// TIA Portal V19 export
DATA_BLOCK "Panel"   // DB1070
{ S7_Optimized_Access := 'TRUE' }
// stored: AutoNumber false, MemoryReserve 100
   VAR RETAIN
      IW : Struct   // Analogwerte
         "LF_CM01.BN01" : Real;   // Leitfähigkeit Bypass Filterpumpe
         "LF_CM01.BN02" : Real;   // Leitfähigkeit Düsen Umwälzung
         "LF_CM02.BN03" : Real;   // Leitfähigkeit Bypass Filterpumpe
         "LF_CM02.BN04" : Real;   // Leitfähigkeit Düsen Umwälzung
         "p_HQ01.BP01" : Real;   // Druck Beutelfiltergehäuse
         "p_HQ02.BP02" : Real;   // Druck Beutelfiltergehäuse
         "p_CM01.BP03" : Real;   // Druck Filterpumpe
         "p_CM01.BP04" : Real;   // Druck Umwälzpumpe
         "p_CM03.BP05" : Real;   // Druck Umwäzpumpe
         "p_CM02.BP06" : Real;   // Druck Filterpumpe
         "p_CM02.BP07" : Real;   // Druck Umwälzpumpe
         "p_CM04.BP08" : Real;   // Druck Umwäzpumpe
         "p_CM05.BP09" : Real;   // Druck Pumpe Entleerung Sammeltank
         "Dfl_GP01.BF01" : Real;   // Durchfluss Versorgung Frischsäure
         "Dfl_GP02.BF02" : Real;   // Durchfluss Entsorgung Altsäure
         "Niv_GP01.BL30" : Real;   // Füllstand Versorgung Frischsäure
         "Niv_GP02.BL31" : Real;   // Füllstand Entsorgung Altsäure
         pH_BE : Real;   // SRM_Auf_BG-QM43
      END_STRUCT;
      Deckel : Struct   // Deckel Säurebecken
         CM01 : Struct
            Auto : Bool;
            Hand : Bool;
            Tipp : Bool;
            links_auf : Bool;
            links_zu : Bool;
            rechts_auf : Bool;
            rechts_zu : Bool;
            SRM_links_auf : Bool;
            SRM_links_zu : Bool;
            SRM_rechts_auf : Bool;
            SRM_rechts_zu : Bool;
            S_links_auf : Bool;   // CM01.BG01
            S_links_zu : Bool;   // CM01.BG02
            S_rechts_auf : Bool;   // CM01.BG03
            S_rechts_zu : Bool;   // CM01.BG04
            Ist_Pos_links : Int;   // 0% = auf; 100% = zu
            Ist_Pos_rechts : Int;   // 0% = auf; 100% = zu
         END_STRUCT;
         CM02 : Struct
            Auto : Bool;
            Hand : Bool;
            Tipp : Bool;
            links_auf : Bool;
            links_zu : Bool;
            rechts_auf : Bool;
            rechts_zu : Bool;
            SRM_links_auf : Bool;
            SRM_links_zu : Bool;
            SRM_rechts_auf : Bool;
            SRM_rechts_zu : Bool;
            S_links_auf : Bool;   // CM02.BG01
            S_links_zu : Bool;   // CM02.BG02
            S_rechts_auf : Bool;   // CM02.BG03
            S_rechts_zu : Bool;   // CM02.BG04
            Ist_Pos_links : Int;   // 0% = auf; 100% = zu
            Ist_Pos_rechts : Int;   // 0% = auf; 100% = zu
         END_STRUCT;
      END_STRUCT;
      RT : Struct   // Schnelllauftor
         K_Auto : Bool;   // Knauf Auto
         T_auf : Bool;   // Taste RT auf
         T_zu : Bool;   // Taste RT zu
         MSS_ok : Bool;   // Motorschutzschalter o.k.
         S_offen : Bool;   // Schnelllauftor offen
         S_geschlossen : Bool;   // Schnelllauftor geschlossen
         ok : Bool;   // Schnelllauftor o.k.
         Status : USInt;
      END_STRUCT;
      Ventilator : Struct   // FU[7]
         Ein : Bool;
         Auto : Bool;
         laeuft : Bool;
         betriebsbereit : Bool;
         Stoerung : Bool;
         Status : USInt;
         SW_Hand : Int;   // [%]
         SW_Auto_AZ : Int;   // [%]
         SW_Auto_aAZ : Int;   // [%]
         speed : Int;   // [%]
      END_STRUCT;
      CM01 : Struct   // HF-Becken 1
         Betrieb : Bool;
         Wartung : Bool;
         Niv_TGS : Bool;   // BL04
         Niv_Min : Bool;   // BL03
         Niv_max : Bool;   // BL02
         Niv_Uel : Bool;   // BL01
         NSP_Auto : Bool;
         GW_LF_FP : Bool;   // BN01
         GW_LF_UP : Bool;   // BN02
         GW_p_FP : Bool;   // BP03
         GW_p_UP : Bool;   // BP04
         Niv_Proz : USInt;
         Sollwert_LF : Real;   // Dosierung
         Dosierung_LF : Bool;   // 0 = WT, 1= LF
      END_STRUCT;
      CM02 : Struct   // HF-Becken 2
         Betrieb : Bool;
         Wartung : Bool;
         Niv_TGS : Bool;   // BL11
         Niv_Min : Bool;   // BL10
         Niv_max : Bool;   // BL09
         Niv_Uel : Bool;   // BL08
         NSP_Auto : Bool;
         GW_LF_FP : Bool;   // BN03
         GW_LF_UP : Bool;   // BN04
         GW_p_FP : Bool;   // BP06
         GW_p_UP : Bool;   // BP07
         Niv_Proz : USInt;
         Sollwert_LF : Real;   // Dosierung
         Dosierung_LF : Bool;   // 0 = WT, 1= LF
      END_STRUCT;
      CM03 : Struct   // Spülbecken 1
         Betrieb : Bool;
         Wartung : Bool;
         Niv_TGS : Bool;   // BL07
         Niv_Min : Bool;   // BL06
         GW_p_UP : Bool;   // BP05
         Niv_Proz : USInt;
         SPR_Auto : Bool;
         SPR_Start_Test : Bool;
         SPR_Stopp_Test : Bool;
         SPR_Zeit_Test : Int;
      END_STRUCT;
      CM04 : Struct   // Spülbecken 2
         Betrieb : Bool;
         Wartung : Bool;
         Niv_TGS : Bool;   // BL14
         Niv_Min : Bool;   // BL13
         GW_p_UP : Bool;   // BP08
         Niv_Proz : USInt;
         SPR_Auto : Bool;
         SPR_Start_Test : Bool;
         SPR_Stopp_Test : Bool;
         SPR_Zeit_Test : Int;
         NSP_Auto : Bool;
         NSP_Zeit : Int;   // pro Korb
         NSP_Start_Test : Bool;
         NSP_Stopp_Test : Bool;
         NSP_Zeit_Tes : Int;
      END_STRUCT;
      CM05 : Struct   // Abwassersammler
         Betrieb : Bool;
         Wartung : Bool;
         Niv_TGS : Bool;   // BL03
         Niv_Min : Bool;   // BL02
         Niv_max : Bool;   // BL01
         Niv_Uel : Bool;   // BL05
         AWA_Bereit : Bool;
         Frg_Abpumpen : Bool;
         GW_p_Pu : Bool;   // BP09
         Niv_Proz : USInt;
      END_STRUCT;
      HQ01 : Struct   // Filtereinheit
         Niv_Leckage : Bool;   // BL05
         GW_p_FG : Bool;   // BP01
         S_FG_zu : Bool;   // BG06
         S_Dkl_FG_li : Bool;   // BG07
         S_Dkl_FG_re : Bool;   // BG08
         Quitt_FW : Bool;
         Quitt_FW_erlaubt : Bool;
         WarnGr_FW : Real;
         Wechsel_FW : Real;
      END_STRUCT;
      HQ02 : Struct   // Filtereinheit
         Niv_Leckage : Bool;   // BL12
         GW_p_FG : Bool;   // BP02
         S_FG_zu : Bool;   // BG09
         S_Dkl_FG_li : Bool;   // BG10
         S_Dkl_FG_re : Bool;   // BG1
         Quitt_FW : Bool;
         Quitt_FW_erlaubt : Bool;
         WarnGr_FW : Real;
         Wechsel_FW : Real;
      END_STRUCT;
      GP01 : Struct   // HF-Versorgung
         Versorgung : Bool;
         Entsorgung : Bool;
         Niv_leer : Bool;   // BL17
         Niv_max : Bool;   // BL20
         IBC_vorhanden : Bool;   // BG21
         Tür_zu_vorn : Bool;   // BG44
         Tür_zu_seitlich : Bool;   // BG43
         LS_PuSu : Bool;   // BL18
         LS_Pumpe : Bool;   // BL15
         LS_Doppelrohr_BL19 : Bool;   // BL19
         LS_PFA_Übergang : Bool;   // BL16
         LS_Uml_Tunnel : Bool;   // BL34
         Niv_Proz : USInt;
         Status : USInt;
      END_STRUCT;
      GP02 : Struct   // HF-Entsorgung
         Versorgung : Bool;
         Entsorgung : Bool;
         Niv_leer : Bool;   // BL24
         Niv_max : Bool;   // BL23
         IBC_vorhanden : Bool;   // BG22
         Tür_zu_seitlich : Bool;   // BG45
         LS_PuSu : Bool;   // BL18
         LS_Pumpe : Bool;   // BL27
         LS_PFA_Übergang : Bool;   // BL25
         LS_Doppelrohr_BL26 : Bool;   // BL26
         LS_Doppelschlauch_BL32 : Bool;   // BL32
         LS_Doppelschlauch_BL33 : Bool;   // BL33
         Niv_Proz : USInt;
         Status : USInt;
      END_STRUCT;
      Havarie_GP0x : Struct
         Soll_Spuelen_CM0x : Real;   // [l]
         Ist_Spuelen_CM0x : Real;   // [l]
      END_STRUCT;
      CL0x : Struct
         "LS_CL01.BL28" : Bool;   // Leckage OK Übergabestation CL01 CL01.BL28
         "LS_CL02.BL29" : Bool;   // Leckage OK Pumpensumpf Säurebecken CL02 CL02.BL29
         Niv_Proz_CL01 : USInt;
         Niv_Proz_CL02 : USInt;
      END_STRUCT;
      FP_CM01 : Struct   // GP01
         Ein : Bool;
         Auto : Bool;
         Bedienung_Erlaubt : Bool;
         betriebsbereit : Bool;
         Stoerung : Bool;
         Sp_Ventil : Struct
            Sollzeit : Int;   // [s]
            Restzeit : Int;   // [s]
         END_STRUCT;
         Sp_Filter : Struct
            Zeit_leeren_Saure : Int;   // [s]
            Zeit_leeren_CM05 : Int;
            Zeit_Spülen : Int;   // [s]
            Wartezeit : Int;   // [s]
            Zeit_füllen : Int;   // [s]
            Restzeit : Int;   // [s]
         END_STRUCT;
         Drucktest_Pumpe : Struct
            Solldruck : Real;
            Sollzeit : Int;
            Restzeit : Int;
            Schritt : USInt;
         END_STRUCT;
         Drucktest_Filter : Struct
            Solldruck : Real;
            Sollzeit : Int;
            Restzeit : Int;
            Schritt : USInt;
         END_STRUCT;
         BA : USInt;   // 0=normal, 1=Filterwechsel, 2=Spülen
         Status : USInt;
         Status_FW : USInt;
         SW_Hand : Int;   // [%]
         SW_Auto_AZ : Int;   // [%]
         SW_Auto_aAZ : Int;   // [%]
         speed : Int;   // [%]
      END_STRUCT;
      UP_CM01 : Struct   // GP02
         Ein : Bool;
         Auto : Bool;
         Bedienung_Erlaubt : Bool;
         betriebsbereit : Bool;
         Stoerung : Bool;
         Sp_Ventil : Struct
            Sollzeit : Int;   // [s]
            Restzeit : Int;   // [s]
         END_STRUCT;
         Drucktest : Struct
            Solldruck : Real;
            Sollzeit : Int;
            Restzeit : Int;
            Schritt : USInt;
         END_STRUCT;
         BA : USInt;   // 0=normal, 1=Ents GP02, 2= Ents GP01, 3=Ents. CM05, 4=Spülen
         Status : USInt;
         SW_Hand : Int;   // [%]
         SW_Auto_AZ : Int;   // [%]
         SW_Auto_aAZ : Int;   // [%]
         speed : Int;   // [%]
      END_STRUCT;
      UP_CM03 : Struct   // GP03
         Ein : Bool;
         Auto : Bool;
         betriebsbereit : Bool;
         Bedienung_Erlaubt : Bool;
         Stoerung : Bool;
         Sp_Ventil : Struct
            Sollzeit : Int;   // [s]
            Restzeit : Int;   // [s]
         END_STRUCT;
         Drucktest : Struct
            Solldruck : Real;
            Sollzeit : Int;
            Restzeit : Int;
            Schritt : USInt;
         END_STRUCT;
         BA : USInt;   // 0=normal, 1=Ents. CM05, 2=Spülen
         Status : USInt;
         SW_Hand : Int;   // [%]
         SW_Auto_AZ : Int;   // [%]
         SW_Auto_aAZ : Int;   // [%]
         speed : Int;   // [%]
      END_STRUCT;
      FP_CM02 : Struct   // GP04
         Ein : Bool;
         Auto : Bool;
         Bedienung_Erlaubt : Bool;
         betriebsbereit : Bool;
         Stoerung : Bool;
         Sp_Ventil : Struct
            Sollzeit : Int;   // [s]
            Restzeit : Int;   // [s]
         END_STRUCT;
         Sp_Filter : Struct
            Zeit_leeren_Saure : Int;   // [s]
            Zeit_leeren_CM05 : Int;
            Zeit_Spülen : Int;   // [s]
            Wartezeit : Int;   // [s]
            Zeit_füllen : Int;   // [s]
            Restzeit : Int;   // [s]
         END_STRUCT;
         Drucktest_Pumpe : Struct
            Solldruck : Real;
            Sollzeit : Int;
            Restzeit : Int;
            Schritt : USInt;
         END_STRUCT;
         Drucktest_Filter : Struct
            Solldruck : Real;
            Sollzeit : Int;
            Restzeit : Int;
            Schritt : USInt;
         END_STRUCT;
         BA : USInt;   // 0=normal, 1=Filterwechse, 2=Spülen
         Status : USInt;
         Status_FW : USInt;
         SW_Hand : Int;   // [%]
         SW_Auto_AZ : Int;   // [%]
         SW_Auto_aAZ : Int;   // [%]
         speed : Int;   // [%]
      END_STRUCT;
      UP_CM02 : Struct   // GP05
         Ein : Bool;
         Auto : Bool;
         Bedienung_Erlaubt : Bool;
         betriebsbereit : Bool;
         Stoerung : Bool;
         Sp_Ventil : Struct
            Sollzeit : Int;   // [s]
            Restzeit : Int;   // [s]
         END_STRUCT;
         Drucktest : Struct
            Solldruck : Real;
            Sollzeit : Int;
            Restzeit : Int;
            Schritt : USInt;
         END_STRUCT;
         BA : USInt;   // 0=normal, 1=Ents GP02, 2= Ents GP01, 3=Ents. CM05, 4=Spülen
         Status : USInt;
         SW_Hand : Int;   // [%]
         SW_Auto_AZ : Int;   // [%]
         SW_Auto_aAZ : Int;   // [%]
         speed : Int;   // [%]
      END_STRUCT;
      UP_CM04 : Struct   // GP06
         Ein : Bool;
         Auto : Bool;
         betriebsbereit : Bool;
         Bedienung_Erlaubt : Bool;
         Stoerung : Bool;
         Sp_Ventil : Struct
            Sollzeit : Int;   // [s]
            Restzeit : Int;   // [s]
         END_STRUCT;
         Drucktest : Struct
            Solldruck : Real;
            Sollzeit : Int;
            Restzeit : Int;
            Schritt : USInt;
         END_STRUCT;
         BA : USInt;   // 0=normal, 1=Ents. CM05, 2=Spülen
         Status : USInt;
         SW_Hand : Int;   // [%]
         SW_Auto_AZ : Int;   // [%]
         SW_Auto_aAZ : Int;   // [%]
         speed : Int;   // [%]
      END_STRUCT;
      Pu_CM05 : Struct   // GP11
         Ein : Bool;
         Auto : Bool;
         Bedienung_Erlaubt : Bool;
         Sp_Ventil : Struct
            Sollzeit : Int;   // [s]
            Restzeit : Int;   // [s]
         END_STRUCT;
         Drucktest : Struct
            Solldruck : Real;
            Sollzeit : Int;
            Restzeit : Int;
            Schritt : USInt;
         END_STRUCT;
         BA : USInt;   // 0=Entl., 1=Kreislauf, 2=Spülen
         Status : USInt;
      END_STRUCT;
      Pu_CL01 : Struct   // GP08
         Ein : Bool;
         Auto : Bool;
         Bedienung_Erlaubt : Bool;
         Sp_Ventil : Struct
            Sollzeit : Int;   // [s]
            Restzeit : Int;   // [s]
         END_STRUCT;
         BA : USInt;   // 0=Ents. CM05, 1=Spülen
         Status : USInt;
      END_STRUCT;
      Pu_CL02 : Struct   // GP09
         Ein : Bool;
         Auto : Bool;
         Bedienung_Erlaubt : Bool;
         Sp_Ventil : Struct
            Sollzeit : Int;   // [s]
            Restzeit : Int;   // [s]
         END_STRUCT;
         BA : USInt;   // 0=Ents. CM05, 1=Spülen
         Status : USInt;
      END_STRUCT;
      Pu_Entl_GP01 : Struct   // GP12
         Ein : Bool;
         Auto : Bool;
         Bedienung_Erlaubt : Bool;
         Sp_Ventil : Struct
            Sollzeit : Int;   // [s]
            Restzeit : Int;   // [s]
         END_STRUCT;
         BA : USInt;   // 0=Ents. CM05, 1=Spülen
         Status : USInt;
      END_STRUCT;
      Pu_Vers_GP01 : Struct   // GP13
         Ein : Bool;
         Auto : Bool;
         Bedienung_Erlaubt : Bool;
         Sp_Ventil : Struct
            Sollzeit : Int;   // [s]
            Restzeit : Int;   // [s]
         END_STRUCT;
         BA : USInt;   // 0=Vers UVGP01, 1=Ents CM05, 2=Spülen
         Status : USInt;
      END_STRUCT;
      Pu_Entl_GP02 : Struct   // GP07
         Ein : Bool;
         Auto : Bool;
         Bedienung_Erlaubt : Bool;
         Sp_Ventil : Struct
            Sollzeit : Int;   // [s]
            Restzeit : Int;   // [s]
         END_STRUCT;
         BA : USInt;   // 0=Ents. CM05, 1=Spülen
         Status : USInt;
      END_STRUCT;
      Pu_Vers_GP02 : Struct   // GP10
         Ein : Bool;
         Auto : Bool;
         Bedienung_Erlaubt : Bool;
         Sp_Ventil : Struct
            Sollzeit : Int;   // [s]
            Restzeit : Int;   // [s]
         END_STRUCT;
         BA : USInt;   // 0=Vers UVGP01, 1=Ents CM05,2= Spülen
         Status : USInt;
      END_STRUCT;
      Pu_Entleeren : Struct   // GP14
         Ein : Bool;
         Status : USInt;
      END_STRUCT;
      Ventil : Struct   // 0 = Aus, 1= aktiv, 2=Störung
         "CM01.QM18" : USInt;   // Eingang Saugleitung Filterpumpe GP01 Säure 01 CM01.QM18
         "CM01.QM19" : USInt;   // Eingang Spülleitung Filterpumpe GP01 Säure 01 CM01.QM19
         "CM01.QM20" : USInt;   // Eingang Spülleitung Umwälzpumpe GP02 Säure 01 CM01.QM20
         "HQ01.QM21" : USInt;   // EingangSäureleitung Filtereinheit HQ02 Säure 01 CM01.QM21
         "HQ01.LV01" : USInt;   // Entlüftungs-/ Überdruckventil Beutelfilter Säure 01 HQ01.LV01
         "HQ01.QM22" : USInt;   // Eingang Spülleitung Filtereinheit HQ01 Säure 01 HQ01.QM22
         "HQ01.QM23" : USInt;   // Ausgang Säureleitung Filtereinheit HQ01 Säure 01 HQ01.QM23
         "HQ01.QM24" : USInt;   // Ausgang Spülleitung Filtereinheit HQ01 Säure 01 zu Sammeltank HQ01.QM24
         "CM01.QM25" : USInt;   // Eingang Saugleitung Umwälzpumpe GP02 Säure 01 CM01.QM25
         "CM01.QM26" : USInt;   // Ausgang Druckleitung Umwälzpumpe GP02 Säure 01 CM01.QM26
         "CM01.QM27" : USInt;   // Ausgang Spülleitung Umwälzpumpe GP02 Säure 01 zu Sammeltank CM01.QM27
         "CM03.QM33" : USInt;   // Eingang Saugleitung Umwälzpumpe GP03 Spülbecken 1 CM03.QM33
         "CM03.QM34" : USInt;   // Ausgang Druckleitung Umwälzpumpe GP03 Spülbecken 1 CM03.QM34
         "CM03.QM36" : USInt;   // Eingang Spülleitung Umwälzpumpe GP03 Spülbecken 1 CM03.QM36
         "CM03.QM37" : USInt;   // Ausgang Spülleitung Umwälzpumpe GP03 Spülbecken 1 CM03.QM37
         "CM02.QM55" : USInt;   // Eingang Saugleitung Filterpumpe GP04 Säure 02 CM02.QM55
         "CM02.QM56" : USInt;   // Eingang Spülleitung Filterpumpe GP04 Säure 02 CM02.QM56
         "CM02.QM57" : USInt;   // Eingang Spülleitung Umwälzpumpe GP05 Säure 02 CM02.QM57
         "HQ02.QM58" : USInt;   // Eingang Spülleitung Filtereinheit HQ02 Säure 02 CM02.QM58
         "HQ02.LV02" : USInt;   // Entlüftungs-/ Überdruckventil Beutelfilter Säure 02 HQ02.LV02
         "HQ02.QM59" : USInt;   // Eingang Säureleitung Filtereinheit HQ02 Säure 02 HQ02.QM59
         "HQ02.QM60" : USInt;   // Ausgang Säureleitung Filtereinheit HQ02 Säure 02 HQ02.QM60
         "HQ02.QM61" : USInt;   // Ausgang Spülleitung Filtereinheit HQ02 Säure 02 zu Sammeltank HQ02.QM61
         "CM02.QM62" : USInt;   // Eingang Saugleitung Umwälzpumpe GP05 Säure 02 CM02.QM62
         "CM02.QM63" : USInt;   // Ausgang Druckleitung Umwälzpumpe GP05 Säure 02 CM02.QM63
         "CM02.QM64" : USInt;   // Ausgang Spülleitung Umwälzpumpe GP05 Säure 02 zu Sammeltank CM02.QM64
         "CM04.QM72" : USInt;   // Eingang Saugleitung Umwälzpumpe GP06 Spülbecken 2 CM04.QM72
         "CM04.QM73" : USInt;   // Ausgang Druckleitung Umwälzpumpe GP06 Spülbecken 2 CM04.QM73
         "CM04.QM75" : USInt;   // Eingang Spülleitung Umwälzpumpe GP06 Spülbecken 2 CM04.QM75
         "CM04.QM76" : USInt;   // Ausgang Spülleitung Umwälzpumpe GP06 Spülbecken 2 CM04.QM76
         "CM04.QM77" : USInt;   // Frischwasserzufuhr Nachdosierung Spülbecken 2 CM04.QM77
         "CL01.QM51" : USInt;   // Zuleitung VE-Wasser-Spülung Pumpe GP08 CL01.QM51
         "CL02.QM52" : USInt;   // Zuleitung VE-Wasser-Spülung Pumpe GP09 CL02.QM52
         "CM05.QM61" : USInt;   // Saugseite Förderpumpe Entleerung GP11 Sammeltank CM05 CM05.QM61
         "CM05.QM62" : USInt;   // Eingang Spülleitung Förderpumpe GP11 Sammeltank CM05 CM05.QM62
         "CM05.QM63" : USInt;   // Ausgang Spülleitung Förderpumpe GP11 Sammeltank CM05 CM05.QM63
         "CM05.QM64" : USInt;   // Druckseite Förderpumpe Entleerung GP11 Sammeltank CM05 CM05.QM64
         "CM03.QM35" : USInt;   // VE-Wasserleitung Spritzregister Spülbecken 1 CM03.QM35
         "CM04.QM74" : USInt;   // VE-Wasserleitung Spritzregister Spülbecken 2 CM04.QM74
         "GP01.QM14" : USInt;   // PFA Schlauchleitung Anbindung IBC Quick Connect Entsorgung GP01.QM14
         "GP01.QM15" : USInt;   // Eingang Saugleitung Membranpumpe GP13 Versorgung Frischsäure GP01.QM15
         "GP01.QM16" : USInt;   // Eingang Spülleitung Membranpumpe GP13 Versorgung Frischsäure GP01.QM16
         "GP01.QM17" : USInt;   // Ausgang Spülleitung Membranpumpe GP13 Versorgung zu Sammeltank GP01.QM17
         "GP01.QM18" : USInt;   // Ausgang Druckleitung Membranpumpe GP13 Versorgung zu UV-GP01 GP01.QM18
         "GP01.QM19" : USInt;   // Verriegelung UV-GP01 Versorgungsleitung zu Säure CM2 GP01.QM19
         "GP01.QM20" : USInt;   // Verriegelung UV-GP01 Versorgungsleitung zu Säure CM1 GP01.QM20
         "GP01.QM21" : USInt;   // Verriegelung UV-GP01 Versorgungsleitung zur Entsorgung GP02 GP01.QM21
         "GP01.QM22" : USInt;   // Verriegelung UV-GP01 Versorgungsleitung zur Versorgung GP01 GP01.QM22
         "GP01.QM23" : USInt;   // VE-Wasser-Spülung GP12 zu Auffangwanne GP01.QM23
         "GP02.QM37" : USInt;   // VE-Wasser-Ventil Leckagesumpf Entsorgung Altsäure GP02.QM37
         "GP02.QM38" : USInt;   // Eingang Saugleitung Membranpumpe GP10 Versorgung aus GP02 GP02.QM38
         "GP02.QM39" : USInt;   // Eingang Spülleitung Membranpumpe GP10 Versorgung aus GP02 GP02.QM39
         "GP02.QM40" : USInt;   // Ausgang Druckleitung Membranpumpe GP10 zu Sammeltank CM05 GP02.QM40
         "GP02.QM41" : USInt;   // Verriegelung UV-GP02 Versorgungsleitung zu UV-GP01 GP02.QM41
         "GP02.QM42" : USInt;   // Ausgang Spülleitung Membranpumpe GP10 zu Sammeltank CM05 GP02.QM42
         "GP02.QM43" : USInt;   // Verriegelung UV-GP02 Entsorgungsleitung zu Entsorgung GP02 GP02.QM43
         "GP02.QM44" : USInt;   // Verriegelung UV-GP02 Entsorgungsleitung zu Versorgung GP01 GP02.QM44
         "GP02.QM45" : USInt;   // Verriegelung UV-GP02 Entsorgungsleitung von Säurebecken CM01 GP02.QM45
         "GP02.QM46" : USInt;   // Verriegelung UV-GP02 Entsorgungsleitung von Säurebecken CM02 GP02.QM46
      END_STRUCT;
      Betriebsart : Struct
         Tipp : Bool;
         Hand : Bool;
         Automatik : Bool;
         Anzeige : USInt;
      END_STRUCT;
      QF : Struct
         WR02 : Struct
            Auto : Bool;
            Hand : Bool;
            Tipp : Bool;
            T_einfahren : Bool;
            T_ausfahren : Bool;
            S_Pos_Ue : Bool;
            S_Pos_BE : Bool;
            S_BK_vl : Bool;
            S_BK_vr : Bool;
            S_BK_hl : Bool;
            S_BK_hr : Bool;
            A_einfahren : Bool;
            A_ausfahren : Bool;
         END_STRUCT;
         WR03 : Struct
            Auto : Bool;
            Hand : Bool;
            Tipp : Bool;
            T_einfahren : Bool;
            T_ausfahren : Bool;
            S_Pos_Ue : Bool;
            S_Pos_BE : Bool;
            S_BK_vl : Bool;
            S_BK_vr : Bool;
            S_BK_hl : Bool;
            S_BK_hr : Bool;
            A_einfahren : Bool;
            A_ausfahren : Bool;
         END_STRUCT;
         P25_kurz_fertig : Bool;
         P25_lang_fertig : Bool;
         P26_fertig : Bool;
         P27_fertig : Bool;
         P28_fertig : Bool;
         P29_kurz_fertig : Bool;
         P29_lang_fertig : Bool;
         P30_fertig : Bool;
      END_STRUCT;
      TW : Struct
         Knauf_Auto : Bool;
         T_Halt : Bool;
         T_vor : Bool;
         T_rueck : Bool;
         T_heben : Bool;
         T_senken : Bool;
         T_heben_li : Bool;
         T_senken_li : Bool;
         T_heben_re : Bool;
         T_senken_re : Bool;
      END_STRUCT;
      Aufgabe : Struct
         Anf_GO : Bool;   // Beide QF nach aussen
         Freigabe : Bool;   // Datenübernahme
         KS_vl_erlaubt : Bool;   // B/E 1
         KS_vr_erlaubt : Bool;   // B/E 2
         GO_li_erlaubt : Bool;   // B/E 3
         GO_re_erlaubt : Bool;   // B/E 4
         KS_hl_erlaubt : Bool;   // B/E 5
         KS_hr_erlaubt : Bool;   // B/E 6
         LS_v_erlaubt : Bool;   // B/E 1
         LS_h_erlaubt : Bool;   // B/E 5
      END_STRUCT;
      Betriebsmodus : Struct
         Normal : Bool;
         Kombi : Bool;
         Wechsel_erlaubt : Bool;
         Korb_151 : Bool;
         Korb_161 : Bool;
         Anzeige : USInt;
      END_STRUCT;
   END_VAR
BEGIN
END_DATA_BLOCK
